FUNCTION_BLOCK FB_DevStateDiagnosis
VAR CONSTANT
	uiFaultMask					:UINT	:=2#0001_1111_1111_0011;	//デバイスエラーのマスク
END_VAR
VAR_IN_OUT
	eEtherCATMaster				:E_EtherCATMaster;	
END_VAR
VAR_OUTPUT
	bError						:BOOL;								//エラー発生を出力
END_VAR
VAR
	uiDevState 			AT%I*	:UINT;								//PDデータとリンク
	
	sMasterName					:STRING;
	
	bErrorState					:ARRAY[0..15] OF BOOL;				//各ステートエラー
	fbBitREdge					:ARRAY[0..15] OF R_TRIG;
	fbMessage					:ARRAY[0..15] OF FB_TcMessage;
	i							:INT;
END_VAR

//マスター名を入力
	IF sMasterName<>TO_STRING(eEtherCATMaster) THEN
		sMasterName:=TO_STRING(eEtherCATMaster);
	END_IF

//エラー状態を出力
	bError:= (uiDevState AND uiFaultMask)<>0 ;

//デバイスの状態チェック、エラーは複数発生する可能性があるので全bitチェック
	FOR i := 0 TO 15 DO
		bErrorState[i]:=(uiDevState AND SHL(1,i))<>0;
	END_FOR

//結果をEventloggerへ
	FOR i := 0 TO 15 BY 1 DO
		fbBitREdge[i](CLK:=bErrorState[i]);
		
		IF fbBitREdge[i].Q THEN
			fbMessage[i].ipArguments.Clear().AddString(sMasterName);
			fbMessage[i].Send();
		END_IF
		
	END_FOR

//FB_Init は常に暗黙的に使用可能で、主に初期化に使用されます。
//戻り値は評価されません。特定の結果を得るために、メソッドを明示的に宣言し、
//そのメソッドに標準の初期化コードをもったコードを追加することができます。戻り値を評価できます。
METHOD FB_Init: BOOL
VAR_INPUT
    bInitRetains: BOOL; // TRUE: 保持変数は初期化されます (ウォーム リセット、あるいはコールド リセット)
    bInCopyCode: BOOL;  // TRUE: 後でコードをコピーする (オンライン変更) ために、インスタンスをコピーします。
END_VAR
fbMessage[0].CreateEx(TC_EVENTS.TkEtherCATMasterDiagnosisEventClass.LinkError);
fbMessage[1].CreateEx(TC_EVENTS.TkEtherCATMasterDiagnosisEventClass.IOLockedAfterLinkErrorIOResetRequired);
fbMessage[2].CreateEx(TC_EVENTS.TkEtherCATMasterDiagnosisEventClass.LinkErrorRedundancyAdapter);
fbMessage[3].CreateEx(TC_EVENTS.TkEtherCATMasterDiagnosisEventClass.MissingOneFrameRedundancyAdapter);
fbMessage[4].CreateEx(TC_EVENTS.TkEtherCATMasterDiagnosisEventClass.OutOfSendResourcesIOResetRequired);
fbMessage[5].CreateEx(TC_EVENTS.TkEtherCATMasterDiagnosisEventClass.WatchdogTriggered);
fbMessage[6].CreateEx(TC_EVENTS.TkEtherCATMasterDiagnosisEventClass.EthernetDriverMiniportNotFound);
fbMessage[7].CreateEx(TC_EVENTS.TkEtherCATMasterDiagnosisEventClass.IOResetActive);
fbMessage[8].CreateEx(TC_EVENTS.TkEtherCATMasterDiagnosisEventClass.AtLeastOneDeviceInINITState);
fbMessage[9].CreateEx(TC_EVENTS.TkEtherCATMasterDiagnosisEventClass.AtLeastOneDeviceInPREOPState);
fbMessage[10].CreateEx(TC_EVENTS.TkEtherCATMasterDiagnosisEventClass.AtLeastOneDeviceInSAFEOPState);
fbMessage[11].CreateEx(TC_EVENTS.TkEtherCATMasterDiagnosisEventClass.AtLeastOneDeviceInERRORState);
fbMessage[12].CreateEx(TC_EVENTS.TkEtherCATMasterDiagnosisEventClass.DCNotInSync);
END_METHOD

END_FUNCTION_BLOCK

(* stored: Version 1.1.0.1, ProductVersion 3.1.4026.18
   POU FB_DevStateDiagnosis: Id {190b1782-5ec4-420d-87aa-52e460bf38f7}, SpecialFunc None
   Method FB_Init: Id {ad34bf28-1a76-4365-abd3-4c1d351cebcd} *)
